FUNCTION_BLOCK FB_ServoAxis ////Blok funkcyjny obslugujacy kompleksowao jedna Os 
VAR_INPUT	
	stSettings				: ST_Axis_Settings;
	bEmergencyStop 			: BOOL;			// Emergency stop pressed	
	bSTO_Signal 			: BOOL;			// STO signal activated

	lrMarkingPos_mm			: LREAL;
	I_TimeTableRef			: I_TimeTable255;
	sTTRowPreambule			: STRING;
	bELM_ChB				: BOOL;
END_VAR
VAR_OUTPUT
	nActEvent					: nAxis_ErrorList;
	udiActErrorCode				: UDINT;
	bBasePosRefreshWarning		: BOOL;
END_VAR
VAR
	fbHomeSensorRTRIG			:R_TRIG;
	iCurrentPositionNumber		:USINT;
	bMoveAbsDone				:BOOL;
	bMoveModuloDone				:BOOL;
	bQuickHomingDone			:BOOL;
	bQuickHomingRequest			:BOOL;
	//OLD
	stInOuts					: st_Axis_InOuts;
	bEnableMotion				: BOOL;		// When TRUE - try to enable axis, when FALSE disable power - safeState
	McPower 					: MC_Power;
	McReset 					: MC_Reset;
	McStop	 					: MC_Stop;
	McMoveAbs 					: MC_MoveAbsolute;
	McMoveModulo				: MC_MoveModulo;
	McMoveRel 					: MC_MoveRelative;
	McMoveVelocity	 			: MC_MoveVelocity;
	McJog	 					: MC_Jog;
	McReadActualPosition	 	: MC_ReadActualPosition;
	McReadActualVelocity	 	: MC_ReadActualVelocity;
	McHome						: MC_Home;
	McBrakeCtrl					: FB_BrakeControl;
	McTorqueMonitor				: FB_TorqueMonitoringEL_Ex2;
	McTorqueCtrl				: MC_TorqueControl;
	stHomimgParams				: ST_HomingOptions;
	fbTOF_Accelerating: TOF;
	bLimitSwitchMin: BOOL;
	bLimitSwitchMax: BOOL;
	iWorkStep_Axis: INT;
	fbFTrig_EmergStop: F_TRIG;
	fbTON_WorkStepTimeout: TON;
	bAlg_Busy, bAlg_Error : BOOL;
	udiAlg_ErrorId	: UDINT;
	fbTON_WorkStepTime_Alg: TON;
	bHP_InHomePos: BOOL;
	udiMcError: UDINT;
	fbTON_ManualJogReset: TON;
	udiErrorCodeToRead: UDINT;
	udiMcErrorToRead: UDINT;
	fbRTRIG_ManGoForward: R_TRIG;
	bOnlySafeState: BOOL;
	bHMI_Plus, bHMI_Minus: BOOL;
	bResetTmr: BOOL;
	bSetNewBrakeCtrl: BOOL;
	nAct_BrakeMode, nNew_BrakeMode: nHP_Axis_BrakeMode;
	fbFTRIG_BreakCtrlDone: F_TRIG;
	bTooglePowerState: BOOL;
	fbRTRIG_ManMoveSwitchSlower: R_TRIG;
	astErrorHistory: ARRAY [1..10] OF stErrorHistoryRow;
	i:USINT;
	lrPosition:LREAL;
	bCircularPositionsSet:BOOL;
END_VAR
VAR PERSISTENT
	lrReferencePositionAtHomeSensor: LREAL:=-1.0;
	lrLastPositionAtHomeSensor:LREAL:=-1.0;
END_VAR
VAR CONSTANT
	NUMBER_OF_PRESET_POSITIONS: USINT:=8;
END_VAR


// Read drive data
stInOuts.stAxis_Data.ReadStatus();
McReadActualPosition(Axis := stInOuts.stAxis_Data, Enable := TRUE);
McReadActualVelocity(Axis := stInOuts.stAxis_Data, Enable := TRUE);

iCurrentPositionNumber := 0;
IF IsHomed AND pIsNotMoving THEN
	FOR i:=1 TO NUMBER_OF_PRESET_POSITIONS DO
		IF ABS(stSettings.arrPositions[i] - ActualPosition) <= stSettings.lrPositionTolerance THEN
			iCurrentPositionNumber := i;
			EXIT;
		END_IF
	END_FOR
END_IF

//Read FB status
ACT_AxisFBs(); 	
ACT_AxisWorkSteps();
//ACT_AxisFBs(); 


fbHomeSensorRTRIG(CLK:=stInOuts.bHomingSensor);
IF stSettings.bEN_CircularPositions AND NOT bCircularPositionsSet THEN
	lrPosition := 0.0;
	FOR i:=1 TO NUMBER_OF_PRESET_POSITIONS DO
		stSettings.arrPositions[i] := lrPosition;
		lrPosition := lrPosition + 360.0/NUMBER_OF_PRESET_POSITIONS;
	END_FOR
	bCircularPositionsSet:=TRUE;
END_IF


IF stSettings.bEN_QuickHoming AND IsHomed AND fbHomeSensorRTRIG.Q THEN
	mSavePositionAtHomeSensor();
	IF lrReferencePositionAtHomeSensor = -1.0 THEN
		lrReferencePositionAtHomeSensor := lrLastPositionAtHomeSensor;
	ELSE
		bQuickHomingRequest := TRUE;
	END_IF
END_IF


IF IsReady AND bQuickHomingRequest THEN
	mQuickHoming();
END_IF

ACTION ACT_AxisFBs:

// Power ON
IF NOT bELM_ChB THEN
	bLimitSwitchMin	:= NOT stInOuts.wI_DriveInfodata.0;
	bLimitSwitchMax	:= NOT stInOuts.wI_DriveInfodata.1;	
ELSE
	bLimitSwitchMin	:= NOT stInOuts.wI_DriveInfodata.8;
	bLimitSwitchMax	:= NOT stInOuts.wI_DriveInfodata.9;	
END_IF
McPower(Axis:=stInOuts.stAxis_Data, Enable:=, Enable_Positive:=NOT bLimitSwitchMax, Enable_Negative:= (NOT bLimitSwitchMin OR McHome.Active));

// Error reset
McReset(Axis:=stInOuts.stAxis_Data);

// Homing
McHome(Axis := stInOuts.stAxis_Data, bCalibrationCam := bLimitSwitchMin, Options := stHomimgParams);

// Stop FBs
McStop(Axis := stInOuts.stAxis_Data, Deceleration := 15000, Jerk := 100000);
McBrakeCtrl(Axis := stInOuts.stAxis_Data);
fbFTRIG_BreakCtrlDone(CLK:= McBrakeCtrl.Busy);
IF fbFTRIG_BreakCtrlDone.Q THEN
	IF McBrakeCtrl.Mode = eBrakeMode_Automatic THEN	nAct_BrakeMode := nHP_Axis_BrakeMode.BrakeMode_Automatic;
	ELSIF McBrakeCtrl.Mode = eBrakeMode_Lock THEN nAct_BrakeMode := nHP_Axis_BrakeMode.BrakeMode_Lock;
	ELSIF McBrakeCtrl.Mode = eBrakeMode_Unlock THEN nAct_BrakeMode := nHP_Axis_BrakeMode.BrakeMode_Unlock;
	END_IF
END_IF
McBrakeCtrl.Execute := FALSE;
// Motion FBs

McJog(Axis := stInOuts.stAxis_Data, Mode := MC_JOGMODE_CONTINOUS, Acceleration := stSettings.rAcceleration, Deceleration := stSettings.rDeceleration, Jerk := 100000);
McMoveAbs(Axis := stInOuts.stAxis_Data, Acceleration := stSettings.rAcceleration, Deceleration := stSettings.rDeceleration, Jerk := 100000);
McMoveRel(Axis := stInOuts.stAxis_Data, Acceleration := stSettings.rAcceleration, Deceleration := stSettings.rDeceleration, Jerk := 100000);
McMoveVelocity(Axis := stInOuts.stAxis_Data, Acceleration := stSettings.rAcceleration, Deceleration := stSettings.rDeceleration, Jerk := 100000);
McMoveModulo(Axis := stInOuts.stAxis_Data, Acceleration := stSettings.rAcceleration, Deceleration := stSettings.rDeceleration, Jerk := 100000, Direction:= MC_Direction.MC_Positive_Direction);
// Torque limitation
McTorqueMonitor( bCalculate:= bSTO_Signal,
	rTorqueLimit:= ,
	Axis:= stInOuts.stAxis_Data);
McTorqueCtrl(Axis := stInOuts.stAxis_Data, Relative := FALSE, ContinuousUpdate := TRUE, TorqueRamp := 100);
END_ACTION

ACTION ACT_AxisWorkSteps:

fbFTrig_EmergStop(CLK:= bEmergencyStop);
IF fbFTrig_EmergStop.Q THEN
	iWorkStep_Axis := 90;
END_IF
IF NOT bEmergencyStop AND iWorkStep_Axis < 90 THEN
	mNewEvent(nEvent := nHP_Axis_ErrorList.STO_SignalActive, ErrorCode:= 0);
	bOnlySafeState := FALSE;
ELSIF NOT bEnableMotion AND Enabled AND bEmergencyStop AND iWorkStep_Axis > 5 AND iWorkStep_Axis < 92 THEN		// Regular disable (when opewn workcover)
	iWorkStep_Axis := 92;
END_IF

CASE iWorkStep_Axis OF
	0:	// Inicjalizacja
		McPower.Enable := McReset.Execute := McHome.Execute := McStop.Execute := FALSE;
		McJog.JogForward := McJog.JogBackwards := McMoveAbs.Execute := McMoveRel.Execute := McMoveVelocity.Execute := FALSE; 
		iWorkStep_Axis := 1;
		
	1:	// Sprawdzenie parametrów pracy
		stSettings.rSlowSpeed_mm_s := LIMIT(0.5, stSettings.rSlowSpeed_mm_s, 10);
		stSettings.rFastSpeed_mm_s := LIMIT(50, stSettings.rFastSpeed_mm_s, 320);
		stSettings.rDeceleration := LIMIT(100, stSettings.rDeceleration, 5000);
		stSettings.rAcceleration := LIMIT(100, stSettings.rAcceleration, 5000);
		stSettings.lrMax_Pos := LIMIT(100, stSettings.lrMax_Pos, 300); 
		iWorkStep_Axis := 5;
		
	5: 	// Sprawdzenie gotowości do załączenia
		IF IsErrorActive THEN
			mNewEvent( nEvent := nHP_Axis_ErrorList.MotionFB_Error,ErrorCode:= stInOuts.stAxis_Data.Status.ErrorID);
		END_IF
		IF McPower.Enable THEN
			IF McPower.Status THEN
				iWorkStep_Axis := 10;
			ELSIF McPower.Error THEN
				mNewEvent( nEvent := nHP_Axis_ErrorList.MotionFB_Error,ErrorCode:= McPower.ErrorID);
			END_IF
		ELSE 
			IF bEnableMotion THEN
				bOnlySafeState := FALSE;
				McPower.Enable :=  TRUE;
			END_IF
		END_IF
		
	10:	// Axis ready for new Cmds
		IF IsErrorActive THEN
			mNewEvent( nEvent := nHP_Axis_ErrorList.MotionFB_Error,ErrorCode:= stInOuts.stAxis_Data.Status.ErrorID);
		END_IF
		fbTON_WorkStepTimeout(IN:= FALSE);
		bMoveAbsDone := bQuickHomingRequest:= bMoveModuloDone:=FALSE;
		
	15:	// Manual mode
		IF bResetTmr THEN
			bResetTmr := FALSE;
			fbTON_ManualJogReset(IN:= FALSE);
		END_IF
		fbTON_ManualJogReset(IN:= McJog.Active, PT:= T#250MS);
		IF fbTON_ManualJogReset.Q THEN
			McJog.JogForward := McJog.JogBackwards := FALSE;
		END_IF
		// Breake control
		IF bSetNewBrakeCtrl THEN
			McBrakeCtrl.Mode := nNew_BrakeMode;
			McBrakeCtrl.Execute := TRUE;	
			bSetNewBrakeCtrl := FALSE; 
		// Enable/disable axis
		ELSIF bTooglePowerState THEN
			McPower.Enable := NOT McPower.Enable;
 			bTooglePowerState := FALSE;
		ELSE
			McPower.Enable S= McJog.JogForward OR McJog.JogBackwards;
		END_IF	
	
	20:	// Homing
		IF McHome.Execute THEN
			IF McHome.Done THEN
				fbTON_WorkStepTimeout(IN:= FALSE);
				iWorkStep_Axis := 21;		// Acurate
			ELSIF McHome.Error THEN
				mNewEvent( nEvent := nHP_Axis_ErrorList.MotionFB_Error,ErrorCode:= McHome.ErrorID);
		//	ELSIF NOT McHome.Busy THEN
		//		mNewEvent( nEvent := nHP_Axis_ErrorList.MotionFB_NotBusy,ErrorCode:= 0);
			END_IF
		ELSE 
			McHome.Position := 0;
			McHome. HomingMode := MC_HomingMode.MC_DefaultHoming;
			stHomimgParams.SearchDirection := MC_Direction.MC_Negative_Direction;
			stHomimgParams.SyncDirection := MC_Direction.MC_Positive_Direction;
			stHomimgParams.SearchVelocity := 30.0;
			stHomimgParams.SyncVelocity := 1;
			stHomimgParams.ReferenceMode := E_EncoderReferenceMode.ENCODERREFERENCEMODE_DEFAULt;
			McHome.Execute := TRUE;
		END_IF
			
	21:	// Home done
		fbTON_WorkStepTimeout(IN:= TRUE,PT:=T#100MS);
		IF fbTON_WorkStepTimeout.Q THEN
			McHome.Execute := FALSE;
			iWorkStep_Axis := 10;	
		END_IF
		
	30:	// Move to absolute position
		McMoveAbs.Execute := TRUE;
		IF McMoveAbs.Busy THEN
			iWorkStep_Axis := 31;		// Done
		ELSIF McMoveAbs.Error THEN
			mNewEvent(nEvent := nHP_Axis_ErrorList.MotionFB_Error, ErrorCode:= McMoveAbs.ErrorID);
		END_IF
	
	31:	// Move ABS done
		IF 	McMoveAbs.Done THEN
			iWorkStep_Axis := 10;	
			bMoveAbsDone := TRUE;
		ELSIF McMoveAbs.Error THEN
			mNewEvent(nEvent := nHP_Axis_ErrorList.MotionFB_Error, ErrorCode:= McMoveAbs.ErrorID);
		END_IF
		
		
	40: //Quick Homing
		bQuickHomingRequest:=FALSE;
		McHome.Execute := TRUE;
		IF McHome.Busy THEN
			fbTON_WorkStepTimeout(IN:= FALSE);
			iWorkStep_Axis := 41;
		ELSIF McHome.Error THEN
			mNewEvent( nEvent := nHP_Axis_ErrorList.MotionFB_Error,ErrorCode:= McHome.ErrorID);
		END_IF
		
	41: //Quick Homing Done
		IF 	McHome.Done THEN
			iWorkStep_Axis := 10;	
			bQuickHomingDone := TRUE;
		ELSIF McHome.Error THEN
			mNewEvent(nEvent := nHP_Axis_ErrorList.MotionFB_Error, ErrorCode:= McHome.ErrorID);
		END_IF
	
	50:	// Move Modulo
		McMoveModulo.Execute := TRUE;
		IF McMoveModulo.Busy THEN
			iWorkStep_Axis := 51;		// Done
		ELSIF McMoveModulo.Error THEN
			mNewEvent(nEvent := nHP_Axis_ErrorList.MotionFB_Error, ErrorCode:= McMoveModulo.ErrorID);
		END_IF
	
	51:	// Move Modulo Done
		IF 	McMoveModulo.Done THEN
			iWorkStep_Axis := 10;	
			bMoveModuloDone := TRUE;
		ELSIF McMoveAbs.Error THEN
			mNewEvent(nEvent := nHP_Axis_ErrorList.MotionFB_Error, ErrorCode:= McMoveModulo.ErrorID);
		END_IF
		
	
	90:	// Go to Safe position
		McMoveVelocity.Execute := McMoveAbs.Execute := McMoveRel.Execute := McStop.Execute := FALSE;
		iWorkStep_Axis := 92;		// Domyślnie tylko wyłącz napęd

	
	92:	// Stop drive and disable power
		IF McStop.Execute THEN
			IF McStop.Done OR NOT Enabled OR McStop.Error THEN	// Disable axis - cant do anything
				McStop.Execute := FALSE;
				McPower.Enable := FALSE;
				IF bOnlySafeState THEN
					bOnlySafeState := FALSE;				
					iWorkStep_Axis := 5;	
				ELSE
					iWorkStep_Axis := 94;	
				END_IF

			END_IF
		ELSE 
			IF Enabled THEN
				McStop.Execute := TRUE;
			ELSE
				IF bOnlySafeState THEN
					bOnlySafeState := FALSE;				
					iWorkStep_Axis := 5;	
				ELSE
					iWorkStep_Axis := 94;	
				END_IF				
			END_IF
		END_IF 
		
	94:	// Axis wait for reset	- NOP
		McReset.Execute := FALSE;
		fbTON_WorkStepTimeout(IN:= FALSE);
	
	95: // Axis reset
		bOnlySafeState := FALSE;
		fbTON_WorkStepTimeout(IN:= TRUE,PT:=T#2S);
		IF McReset.Execute THEN
			IF McReset.Done THEN	// Reset axis
				McReset.Execute := FALSE;
				fbTON_WorkStepTimeout(IN:= FALSE);
				iWorkStep_Axis := 96;
			ELSIF McReset.Error THEN		//NOT McReset.Busy OR 
				McReset.Execute := FALSE;
				iWorkStep_Axis := 97;
			END_IF
		ELSE 
			McHome.Execute := McStop.Execute := McJog.JogForward := McJog.JogBackwards := FALSE;
			McMoveAbs.Execute := McMoveRel.Execute := McMoveVelocity.Execute := FALSE; 
			IF stInOuts.stAxis_Data.Status.Error THEN
				McReset.Execute := TRUE;
			ELSE
				fbTON_WorkStepTimeout(IN:= FALSE);
				iWorkStep_Axis := 96;
			END_IF
		END_IF
		
	96:	// Reset succesfull
		nActEvent := nHP_Axis_ErrorList.NoError;
		fbTON_WorkStepTimeout(IN:= TRUE, PT:= T#40MS);
		IF fbTON_WorkStepTimeout.Q THEN
			fbTON_WorkStepTimeout(IN:= FALSE);
			iWorkStep_Axis := 5;
		END_IF
		
	97:	// Reset error
		nActEvent := nHP_Axis_ErrorList.MotionFB_Error;
		iWorkStep_Axis := 90;	
END_CASE
END_ACTION

PROPERTY ActualPosition : LREAL
GET
IF McReadActualPosition.Valid AND IsHomed THEN		
	ActualPosition := McReadActualPosition.Position;
ELSE
	ActualPosition := -1;
END_IF
END_GET
END_PROPERTY

PROPERTY ActualVelocity : LREAL
GET
IF McReadActualVelocity.Valid THEN
	ActualVelocity := McReadActualVelocity.ActualVelocity;
ELSE
	ActualVelocity := -1;
END_IF
END_GET
END_PROPERTY

PROPERTY Enabled : BOOL
GET
Enabled:= McPower.Status;
END_GET
SET
IF Enabled AND bSTO_Signal THEN
	bEnableMotion := TRUE;	
	McPower.Enable := TRUE;
	ACT_AxisFBs();
ELSE
	IF IsMoving THEN
		mNewEvent( nEvent := nHP_Axis_ErrorList.ProgramError ,ErrorCode:= INT_TO_UDINT(iWorkStep_Axis));	
		bEnableMotion := FALSE;
	ELSE
		bEnableMotion := FALSE;	
		McPower.Enable := FALSE;
		ACT_AxisFBs();
		iWorkStep_Axis := 5;
	END_IF
END_IF
END_SET
END_PROPERTY

PROPERTY IsErrorActive : BOOL
GET
IsErrorActive := stInOuts.stAxis_Data.Status.Error OR iWorkStep_Axis >= 90;
END_GET
END_PROPERTY

PROPERTY IsHomed : BOOL
GET
IsHomed := stInOuts.stAxis_Data.Status.Homed;
END_GET
END_PROPERTY

PROPERTY IsMoving : BOOL
GET
IsMoving := stInOuts.stAxis_Data.Status.Moving;
END_GET
END_PROPERTY

PROPERTY IsReady : BOOL
GET
IsReady := stInOuts.stAxis_Data.Status.Operational AND NOT stInOuts.stAxis_Data.Status.Error AND McPower.Status AND iWorkStep_Axis = 10;
END_GET
END_PROPERTY

PROPERTY IsReadyForOperation : BOOL
GET
IsReadyForOperation := IsReady;
END_GET
END_PROPERTY

METHOD mAddTimeStat : BOOL
VAR_INPUT
	sText 		: STRING(255);
END_VAR
VAR
	sTextTmp	: STRING(255);
END_VAR
IF I_TimeTableRef <> 0 THEN
	CONCAT2(pSrcString1 := ADR(sTTRowPreambule), pSrcString2 := ADR(sText), pDstString := ADR(sTextTmp), nDstSize := SIZEOF(sTextTmp));
	I_TimeTableRef.mPushText(sText := sTextTmp);
END_IF
END_METHOD

PROPERTY ManualMode : BOOL
GET
ManualMode := iWorkStep_Axis = 15;
END_GET
SET
IF ManualMode AND NOT IsErrorActive THEN		
	bEnableMotion := TRUE;	
	McPower.Enable := TRUE;
	ACT_AxisFBs();
	IF Enabled THEN
		iWorkStep_Axis := 15;
	END_IF	
ELSIF NOT ManualMode THEN
	IF iWorkStep_Axis = 15 THEN
		McJog(Axis:= stInOuts.stAxis_Data, JogForward := FALSE, JogBackwards := FALSE);
		bEnableMotion := TRUE;	
		McPower.Enable := FALSE;
		McBrakeCtrl.Execute := TRUE;
		McBrakeCtrl.Mode := E_BrakeMode.eBrakeMode_Automatic;
		ACT_AxisFBs();
		iWorkStep_Axis := 5;		
	END_IF
END_IF
END_SET
END_PROPERTY

METHOD mFullHoming : BOOL
VAR_INPUT
END_VAR
VAR_OUTPUT
	bBusy		: BOOL;
	bError		: BOOL;
	udiErrorId	: UDINT;
END_VAR
IF IsReady THEN
	iWorkStep_Axis := 20;
	bBusy := TRUE;
ELSIF iWorkStep_Axis >= 20 AND iWorkStep_Axis <= 24 THEN
	bBusy := McHome.Busy;
	mFullHoming := McHome.Done;
	bError := McHome.Error;
	udiErrorId := McHome.ErrorID;
ELSE
	mFullHoming := TRUE;
	bError := TRUE;
	udiErrorId := INT_TO_UINT(iWorkStep_Axis);	
END_IF
END_METHOD

METHOD mManualMove : BOOL
VAR_INPUT
	bGoUp		: BOOL;
	bGoDown		: BOOL;
	bSlow		: BOOL;
	bFast		: BOOL;
END_VAR
IF bGoUp OR bGoDown THEN
	bHMI_Plus := bHMI_Minus := FALSE;
	fbTON_ManualJogReset(IN:= FALSE);	
END_IF
fbRTRIG_ManGoForward(CLK:= bGoUp OR bHMI_Plus);

IF fbRTRIG_ManMoveSwitchSlower.Q THEN
		McJog(Axis := stInOuts.stAxis_Data, JogBackwards := FALSE, JogForward := FALSE);	
END_IF

IF bSlow THEN
	McJog.JogForward := (bHMI_Plus OR bGoUp) AND NOT bGoDown;
	McJog.JogBackwards := (bHMI_Minus OR bGoDown) AND NOT bGoUp;
ELSIF bFast THEN
	McJog.Velocity := 20;
	McJog.JogForward := bGoUp AND NOT bGoDown;
	McJog.JogBackwards := bGoDown AND NOT bGoUp;
ELSE	
	McJog.Velocity := LIMIT(0.1, stSettings.rSlowSpeed_mm_s/2, 4);
	McJog.JogForward := bHMI_Plus AND NOT bHMI_Minus;
	McJog.JogBackwards := bHMI_Minus AND NOT bHMI_Plus;
END_IF
END_METHOD

METHOD mMoveFastToPresetPos : BOOL
VAR_INPUT
	iPosNumber	:USINT;
	bFast:BOOL;
END_VAR
VAR_OUTPUT
	bBusy		: BOOL;
	bError		: BOOL;
	udiErrorId	: UDINT;
END_VAR
mMoveFastToPresetPos :=FALSE;
IF IsReady THEN
	iPosNumber := MIN(20,iPosNumber);
	McMoveAbs.Position := stSettings.arrPositions[iPosNumber];
	IF bFast THEN
		McMoveAbs.Velocity := LIMIT(10, stSettings.rFastSpeed_mm_s, 320);
	ELSE
		McMoveAbs.Velocity := LIMIT(0.5, stSettings.rSlowSpeed_mm_s, 20);
	END_IF
	iWorkStep_Axis := 30;
ELSIF McMoveAbs.Error OR iWorkStep_Axis <30 OR iWorkStep_Axis >31  THEN
	mMoveFastToPresetPos := TRUE;
	bError := TRUE;
	udiErrorId := INT_TO_UINT(iWorkStep_Axis);	
END_IF

bBusy := McMoveAbs.Busy;
IF bMoveAbsDone THEN
	mMoveFastToPresetPos := TRUE;
	bMoveAbsDone :=FALSE;
END_IF;
END_METHOD

METHOD mMoveModuloToPosition : BOOL
VAR_INPUT
	iPosNumber	:USINT;
	bFast:BOOL;
END_VAR
VAR_OUTPUT
	bBusy		: BOOL;
	bError		: BOOL;
	udiErrorId	: UDINT;
END_VAR
mMoveModuloToPosition :=FALSE;
IF IsReady THEN
	iPosNumber := MIN(20,iPosNumber);
	McMoveModulo.Position := stSettings.arrPositions[iPosNumber];
	IF bFast THEN
		McMoveModulo.Velocity := LIMIT(10, stSettings.rFastSpeed_mm_s, 320);
	ELSE
		McMoveModulo.Velocity := LIMIT(0.5, stSettings.rSlowSpeed_mm_s, 20);
	END_IF
	iWorkStep_Axis := 50;
	McMoveModulo.Execute := TRUE;	
ELSIF McMoveModulo.Error OR iWorkStep_Axis <50 OR iWorkStep_Axis >51  THEN
	mMoveModuloToPosition := TRUE;
	bError := TRUE;
	udiErrorId := INT_TO_UINT(iWorkStep_Axis);	
END_IF

bBusy := McMoveModulo.Busy;
IF bMoveModuloDone THEN
	mMoveModuloToPosition := TRUE;
	bMoveModuloDone :=FALSE;
END_IF;
udiErrorId := McMoveModulo.ErrorID;
END_METHOD

METHOD INTERNAL mNewEvent : BOOL
VAR_INPUT
	nEvent: nAxis_ErrorList;
	ErrorCode: UDINT;
END_VAR

MEMMOVE(srcAddr:= ADR(astErrorHistory[1]), destAddr := ADR(astErrorHistory[2]), n:= 9* SIZEOF(astErrorHistory[1]));
astErrorHistory[1].tTimeStamp := TIME();
astErrorHistory[1].sDescription := TO_STRING(nEvent);
astErrorHistory[1].iWorkStep1 := iWorkStep_Axis;
astErrorHistory[1].udiErrorCode := ErrorCode;

iWorkStep_Axis := 90;
bAlg_Error := TRUE;
udiErrorCodeToRead := udiAlg_ErrorId := nEvent;
nActEvent := nEvent;
udiActErrorCode:= ErrorCode;
fbTON_WorkStepTime_Alg(IN := FALSE);
IF ErrorCode <> 0 THEN
	udiMcErrorToRead := udiMcError:= ErrorCode;
END_IF



McReset.Execute := McHome.Execute := McStop.Execute := FALSE;
McJog.JogForward := McJog.JogBackwards := McMoveAbs.Execute := McMoveRel.Execute := McMoveVelocity.Execute := FALSE;
ACT_AxisFBs();
END_METHOD

METHOD mQuickHoming : BOOL
VAR_INPUT
END_VAR
VAR_OUTPUT
	bBusy		: BOOL;
	bError		: BOOL;
	udiErrorId	: UDINT;
END_VAR
mQuickHoming :=FALSE;
IF IsReady AND lrReferencePositionAtHomeSensor > 0 AND lrLastPositionAtHomeSensor > 0 THEN
	McHome.Position := ActualPosition + (lrReferencePositionAtHomeSensor - lrLastPositionAtHomeSensor);
	McHome. HomingMode := MC_HomingMode.MC_Direct;
	iWorkStep_Axis := 40;
ELSIF McHome.Error OR iWorkStep_Axis <40 OR iWorkStep_Axis >41  THEN
	mQuickHoming := TRUE;
	bError := TRUE;
	udiErrorId := INT_TO_UINT(iWorkStep_Axis);	
END_IF

bBusy := McHome.Busy;
IF bQuickHomingDone THEN
	mQuickHoming := TRUE;
	bQuickHomingDone :=FALSE;
END_IF;
udiErrorId := McHome.ErrorID;
END_METHOD

METHOD mReadError : BOOL
VAR_OUTPUT
	udiErrorID		: UDINT;
	udiMcErrorID	: UDINT;
END_VAR
IF udiErrorCodeToRead <> 0 THEN
	mReadError:= TRUE;
	udiErrorID := udiErrorCodeToRead;
	udiErrorCodeToRead := 0;
END_IF
IF udiMcErrorToRead <> 0 THEN
	mReadError:= TRUE;
	udiMcErrorID := udiMcErrorToRead;
	udiMcErrorToRead := 0;
END_IF
END_METHOD

METHOD mReset : BOOL
VAR_OUTPUT
	bBusy		: BOOL;
	bError		: BOOL;
	udiErrorId	: UDINT;
END_VAR
IF iWorkStep_Axis = 94 THEN
	iWorkStep_Axis := 95;
	bBusy := TRUE;
ELSIF iWorkStep_Axis = 95 THEN
	bBusy := TRUE;
ELSIF iWorkStep_Axis = 96 THEN
	iWorkStep_Axis := 5;
	mReset := TRUE;
ELSIF iWorkStep_Axis = 97 THEN
	mReset := TRUE;
	bError := TRUE;
	udiErrorId := McReset.ErrorID;
ELSIF iWorkStep_Axis = 5 OR iWorkStep_Axis = 10 THEN
	mReset := TRUE; 
END_IF
END_METHOD

METHOD mSavePositionAtHomeSensor : BOOL
VAR_INPUT
END_VAR
IF ActualPosition <> -1 THEN
	lrLastPositionAtHomeSensor:=ActualPosition;
END_IF;
END_METHOD

{attribue 'monitoring':= call}
PROPERTY pCurrentPositionNumber : USINT
GET
pCurrentPositionNumber:=iCurrentPositionNumber;
END_GET
END_PROPERTY

{attribue 'monitoring':= call}
PROPERTY pIsInTargetPosition : BOOL
GET
pIsInTargetPosition := TRUE;
END_GET
END_PROPERTY

{attribue 'monitoring':= call}
PROPERTY pIsNotMoving : BOOL
GET
pIsNotMoving := TRUE;
END_GET
END_PROPERTY

END_FUNCTION_BLOCK

(* stored: Version 1.1.0.1, ProductVersion 3.1.4024.15
   POU FB_ServoAxis: Id {3057f7b8-ac98-4f2d-b555-83dd6c315250}, SpecialFunc None
   Folder Methods: Id {86110dc1-c583-424f-8e1a-53f0e16b101e}
   Folder Properties: Id {8dc25682-5df1-487c-935d-d480b60343c3}
   Action ACT_AxisFBs: Id {1733d200-0c8f-4641-80db-f206791f3515}
   Action ACT_AxisWorkSteps: Id {24332e8c-4fda-4b2a-bd2c-6d7b94bd461c}
   Property ActualPosition: Id {f40194ba-8306-4aaa-b5b5-5fb0758d9b45}
   Get Get: Id {8bac339c-d060-4766-ad8b-fd8c908a3488}
   Property ActualVelocity: Id {ff223880-cd07-4f47-8533-6780d3523a7c}
   Get Get: Id {78818ba6-1efe-447e-8266-54cd48988813}
   Property Enabled: Id {20ee9f61-720c-40a2-84c5-331a0b62253a}
   Get Get: Id {6f777018-1d15-4443-86fe-bcc9014295bc}
   Set Set: Id {aa69c21e-9129-4b1c-ba60-b2116521a411}
   Property IsErrorActive: Id {da3f3089-581e-41ca-8bcd-c78e51817caa}
   Get Get: Id {436b39d5-59d0-48e6-8f59-40a1bc78273a}
   Property IsHomed: Id {f71d9df2-615f-49d5-9f8f-a7959eb3e890}
   Get Get: Id {214f06e1-9c57-412c-bce6-1826f7c03c7d}
   Property IsMoving: Id {d921ac5b-ba42-4853-9806-c4dcb58d889c}
   Get Get: Id {f68ebf89-02ea-47cb-8cf6-53ef2c6e6de6}
   Property IsReady: Id {6e65633e-98e6-41e4-9524-0f21768d5334}
   Get Get: Id {4e0e5a66-9481-4905-b577-efae5ddc6ef5}
   Property IsReadyForOperation: Id {2ddbe4a9-bbca-4d1c-ae6e-6df6b6493cff}
   Get Get: Id {8a0a6e10-abef-4020-8068-05456676117e}
   Method mAddTimeStat: Id {ab5ac6de-4b6f-4492-81c5-0cd32a15380e}
   Property ManualMode: Id {6c92fae3-cad0-41de-951a-c69e4b5af978}
   Get Get: Id {cecf79a4-7b4f-46d1-8871-ee07bc7603c3}
   Set Set: Id {0920975c-0fcd-426c-b9f5-24f77c4a4de2}
   Method mFullHoming: Id {a262032b-63e5-4e87-a4b0-e16a24b03a3b}
   Method mManualMove: Id {3ec3a8b0-e761-4ba5-86e3-9564d84aa78d}
   Method mMoveFastToPresetPos: Id {17b7a812-32ab-4488-9109-06aa0299f113}
   Method mMoveModuloToPosition: Id {b9786ee7-83c2-4602-a755-a5d8da1d53c5}
   Method mNewEvent: Id {45dc65cc-cc78-49f4-a976-6b04a137582d}
   Method mQuickHoming: Id {5b03c9ef-9972-4bbe-81ff-bccad90f604c}
   Method mReadError: Id {0a9a6395-d6a0-4d73-bd08-a80371a337db}
   Method mReset: Id {4c71a6d0-2eb8-4fd5-9ef2-16b78ed57f34}
   Method mSavePositionAtHomeSensor: Id {3a59daed-c1be-449e-8865-4c1bfb4a7379}
   Property pCurrentPositionNumber: Id {ea3d6f95-12cc-4ac1-9e24-d1e623d6380c}
   Get Get: Id {5c223598-c8c8-44d8-8e1f-7aaddfe49b9a}
   Property pIsInTargetPosition: Id {7c58df86-0d69-4a2c-830b-ded4fd793ede}
   Get Get: Id {e786766e-c47f-4a16-8b97-2ac914454196}
   Property pIsNotMoving: Id {55c0575a-37a0-40ed-985f-602114fa2c8e}
   Get Get: Id {cb1572cd-ba6b-409d-8282-8e38c003a699} *)
